Omron CX-Programmer project NewProject (CX-Programmer 9.75)

# PLC NewPLC1: CJ2M CPU11

## Global symbols (name address type ; comment)
0.01 BOOL  ; START
0.02 BOOL  ; STOP
0.03 BOOL  ; S1
0.04 BOOL  ; S2
0.05 BOOL  ; S3
0.08 BOOL  ; S1
1.00 BOOL  ; RUN
1.01 BOOL  ; M1
1.02 BOOL  ; M2
1.03 BOOL  ; M3

## Program NewProgram1 (cyclic task 0)
; CONVEYOR BELT SERIES MOTOR CONTROL

### Section Section1
; LADDER LOGIC PROGRAMMING OMRON PLC

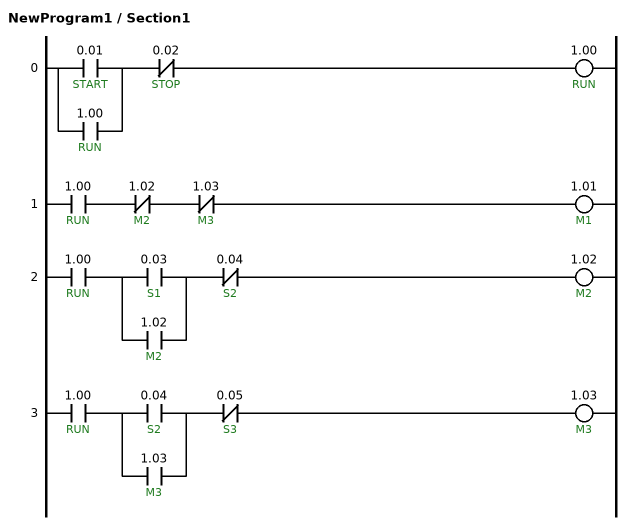
; rung 0
LD 0.01  ; START
OR 1.00  ; RUN
ANDNOT 0.02  ; STOP
OUT 1.00  ; RUN
; rung 1
LD 1.00  ; RUN
ANDNOT 1.02  ; M2
ANDNOT 1.03  ; M3
OUT 1.01  ; M1
; rung 2
LD 1.00  ; RUN
LD 0.03  ; S1
OR 1.02  ; M2
ANDLD
ANDNOT 0.04  ; S2
OUT 1.02  ; M2
; rung 3
LD 1.00  ; RUN
LD 0.04  ; S2
OR 1.03  ; M3
ANDLD
ANDNOT 0.05  ; S3
OUT 1.03  ; M3

### Section END
; rung 0
END(001)